// TIA Portal V20 export
DATA_BLOCK "IDB_FB_Technology"   // DB38
// stored: InstanceOfName ProductionLine.FB_Technology, InstanceOfType FB, Namespace ProductionLine
"ProductionLine.FB_Technology"
   // VAR
   //    IP11 : String;
   //    IP12 : String;
   //    IP21 : String;
   //    IP22 : String;
   //    IP23 : String;
   //    IP31 : String;
   //    IP32 : String;
   //    IP41 : String;
   //    IP42 : String;
   //    ComDownStream : Struct
   //       DP1 : Bool;
   //       DP2 : Bool;
   //       DP3 : Bool;
   //       DP4 : Bool;
   //    END_STRUCT;
   //    ComTimmerDP1 { S7_SetPoint := 'True'} : TON_TIME;
   //    ComTimmerDP2 { S7_SetPoint := 'True'} : TON_TIME;
   //    ComTimmerDP3 { S7_SetPoint := 'True'} : TON_TIME;
   //    ComTimmerDP4 { S7_SetPoint := 'True'} : TON_TIME;
   // END_VAR
BEGIN
END_DATA_BLOCK
